FUNCTION_BLOCK orchestratorFB (* Generated orchestrator *)
  (* Standard: 61499-2 *)
  (* Version 1.0, 2020-10-07, generator *)
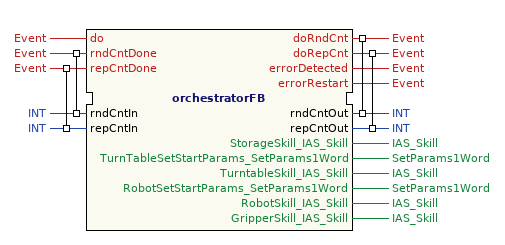
  EVENT_INPUT
    do; (* Start whole process *)
    rndCntDone WITH rndCntIn; (* Whole process (round) counter was updated *)
    repCntDone WITH repCntIn; (* Repetition counter was updated *)
  END_EVENT
  EVENT_OUTPUT
    doRndCnt WITH rndCntOut; (* Update of the whole process (round) counter *)
    doRepCnt WITH repCntOut; (* Update of the repetition counter *)
    errorDetected; (* Triggered when an error signal was received (defined by adapter service sequence) *)
    errorRestart; (* Triggered when error handling and skill restart is started after error signal *)
  END_EVENT
  VAR_INPUT
    rndCntIn : INT; (* Iteration number of the whole process (round) *)
    repCntIn : INT; (* Iteration number of the current repetition process *)
  END_VAR
  VAR_OUTPUT
    rndCntOut : INT; (* Iteration number of the whole process (round) *)
    repCntOut : INT; (* Iteration number of the current repetition process *)
  END_VAR
  PLUGS
    StorageSkill_IAS_Skill : IAS_Skill;
    TurnTableSetStartParams_SetParams1Word : SetParams1Word;
    TurntableSkill_IAS_Skill : IAS_Skill;
    RobotSetStartParams_SetParams1Word : SetParams1Word;
    RobotSkill_IAS_Skill : IAS_Skill;
    GripperSkill_IAS_Skill : IAS_Skill;
  END_PLUGS
  EC_STATES
    START; (* Initial State *)
    Init : round_cnt_reset -> doRndCnt; (* If the adapter of a skill needs an initialization call *)
    Round_Start; (* Start of an iteration of the whole process *)
    Round_End : round_cnt_inc -> doRndCnt; (* End of an iteration of the whole process *)
    0_StorageSkill_Start_0 : -> StorageSkill_IAS_Skill.start;
    1_StorageSkill_RSP_rec_0;
    3_StorageSkill_End_0;
    5_TurnTableSetStartParams_End_1 : 4_TurnTableSetStartParams_Start_1_Alg0 -> TurnTableSetStartParams_SetParams1Word.IND;
    6_TurntableSkill_Start_2 : -> TurntableSkill_IAS_Skill.start;
    7_TurntableSkill_RSP_rec_2;
    9_TurntableSkill_End_2;
    10_StorageSkill_Start_3 : -> StorageSkill_IAS_Skill.start;
    11_StorageSkill_RSP_rec_3;
    13_StorageSkill_End_3;
    15_TurnTableSetStartParams_End_4 : 14_TurnTableSetStartParams_Start_4_Alg1 -> TurnTableSetStartParams_SetParams1Word.IND;
    16_TurntableSkill_Start_5 : -> TurntableSkill_IAS_Skill.start;
    17_TurntableSkill_RSP_rec_5;
    19_TurntableSkill_End_5;
    21_RobotSetStartParams_End_6 : 20_RobotSetStartParams_Start_6_Alg2 -> RobotSetStartParams_SetParams1Word.IND;
    22_RobotSkill_Start_7 : -> RobotSkill_IAS_Skill.start;
    23_RobotSkill_RSP_rec_7;
    25_RobotSkill_End_7;
    26_GripperSkill_Start_8 : -> GripperSkill_IAS_Skill.start;
    27_GripperSkill_RSP_rec_8;
    29_GripperSkill_End_8;
    31_RobotSetStartParams_End_9 : 30_RobotSetStartParams_Start_9_Alg3 -> RobotSetStartParams_SetParams1Word.IND;
    32_RobotSkill_Start_10 : -> RobotSkill_IAS_Skill.start;
    33_RobotSkill_RSP_rec_10;
    35_RobotSkill_End_10;
    36_GripperSkill_Start_11 : -> GripperSkill_IAS_Skill.start;
    37_GripperSkill_RSP_rec_11;
    39_GripperSkill_End_11;
    41_RobotSetStartParams_End_12 : 40_RobotSetStartParams_Start_12_Alg4 -> RobotSetStartParams_SetParams1Word.IND;
    42_RobotSkill_Start_13 : -> RobotSkill_IAS_Skill.start;
    43_RobotSkill_RSP_rec_13;
    45_RobotSkill_End_13;
    46_GripperSkill_Start_14 : -> GripperSkill_IAS_Skill.start;
    47_GripperSkill_RSP_rec_14;
    49_GripperSkill_End_14;
    51_RobotSetStartParams_End_15 : 50_RobotSetStartParams_Start_15_Alg5 -> RobotSetStartParams_SetParams1Word.IND;
    52_RobotSkill_Start_16 : -> RobotSkill_IAS_Skill.start;
    53_RobotSkill_RSP_rec_16;
    55_RobotSkill_End_16;
    56_GripperSkill_Start_17 : -> GripperSkill_IAS_Skill.start;
    57_GripperSkill_RSP_rec_17;
    59_GripperSkill_End_17;
    61_RobotSetStartParams_End_18 : 60_RobotSetStartParams_Start_18_Alg6 -> RobotSetStartParams_SetParams1Word.IND;
    62_RobotSkill_Start_19 : -> RobotSkill_IAS_Skill.start;
    63_RobotSkill_RSP_rec_19;
    65_RobotSkill_End_19;
    66_GripperSkill_Start_20 : -> GripperSkill_IAS_Skill.start;
    67_GripperSkill_RSP_rec_20;
    69_GripperSkill_End_20;
    71_RobotSetStartParams_End_21 : 70_RobotSetStartParams_Start_21_Alg7 -> RobotSetStartParams_SetParams1Word.IND;
    72_RobotSkill_Start_22 : -> RobotSkill_IAS_Skill.start;
    73_RobotSkill_RSP_rec_22;
    75_RobotSkill_End_22;
    76_GripperSkill_Start_23 : -> GripperSkill_IAS_Skill.start;
    77_GripperSkill_RSP_rec_23;
    79_GripperSkill_End_23;
    81_RobotSetStartParams_End_24 : 80_RobotSetStartParams_Start_24_Alg8 -> RobotSetStartParams_SetParams1Word.IND;
    82_RobotSkill_Start_25 : -> RobotSkill_IAS_Skill.start;
    83_RobotSkill_RSP_rec_25;
    85_RobotSkill_End_25;
    86_GripperSkill_Start_26 : -> GripperSkill_IAS_Skill.start;
    87_GripperSkill_RSP_rec_26;
    89_GripperSkill_End_26;
    91_RobotSetStartParams_End_27 : 90_RobotSetStartParams_Start_27_Alg9 -> RobotSetStartParams_SetParams1Word.IND;
    92_RobotSkill_Start_28 : -> RobotSkill_IAS_Skill.start;
    93_RobotSkill_RSP_rec_28;
    95_RobotSkill_End_28;
    96_GripperSkill_Start_29 : -> GripperSkill_IAS_Skill.start;
    97_GripperSkill_RSP_rec_29;
    99_GripperSkill_End_29;
    101_RobotSetStartParams_End_30 : 100_RobotSetStartParams_Start_30_Alg10 -> RobotSetStartParams_SetParams1Word.IND;
    102_RobotSkill_Start_31 : -> RobotSkill_IAS_Skill.start;
    103_RobotSkill_RSP_rec_31;
    105_RobotSkill_End_31;
  END_STATES
  EC_TRANSITIONS
    START TO Init := do;
    Init TO Round_Start := 1;
    Round_End TO Round_Start := do;
    Round_Start TO 0_StorageSkill_Start_0 := 1;
    105_RobotSkill_End_31 TO Round_End := 1;
    0_StorageSkill_Start_0 TO 1_StorageSkill_RSP_rec_0 := StorageSkill_IAS_Skill.RSP[StorageSkill_IAS_Skill.currentState="Executing"];
    1_StorageSkill_RSP_rec_0 TO 3_StorageSkill_End_0 := StorageSkill_IAS_Skill.RSP[StorageSkill_IAS_Skill.currentState="Idle"];
    3_StorageSkill_End_0 TO 5_TurnTableSetStartParams_End_1 := 1;
    5_TurnTableSetStartParams_End_1 TO 6_TurntableSkill_Start_2 := 1;
    6_TurntableSkill_Start_2 TO 7_TurntableSkill_RSP_rec_2 := TurntableSkill_IAS_Skill.RSP[TurntableSkill_IAS_Skill.currentState="Executing"];
    7_TurntableSkill_RSP_rec_2 TO 9_TurntableSkill_End_2 := TurntableSkill_IAS_Skill.RSP[TurntableSkill_IAS_Skill.currentState="Idle"];
    9_TurntableSkill_End_2 TO 10_StorageSkill_Start_3 := 1;
    10_StorageSkill_Start_3 TO 11_StorageSkill_RSP_rec_3 := StorageSkill_IAS_Skill.RSP[StorageSkill_IAS_Skill.currentState="Executing"];
    11_StorageSkill_RSP_rec_3 TO 13_StorageSkill_End_3 := StorageSkill_IAS_Skill.RSP[StorageSkill_IAS_Skill.currentState="Idle"];
    13_StorageSkill_End_3 TO 15_TurnTableSetStartParams_End_4 := 1;
    15_TurnTableSetStartParams_End_4 TO 16_TurntableSkill_Start_5 := 1;
    16_TurntableSkill_Start_5 TO 17_TurntableSkill_RSP_rec_5 := TurntableSkill_IAS_Skill.RSP[TurntableSkill_IAS_Skill.currentState="Executing"];
    17_TurntableSkill_RSP_rec_5 TO 19_TurntableSkill_End_5 := TurntableSkill_IAS_Skill.RSP[TurntableSkill_IAS_Skill.currentState="Idle"];
    19_TurntableSkill_End_5 TO 21_RobotSetStartParams_End_6 := 1;
    21_RobotSetStartParams_End_6 TO 22_RobotSkill_Start_7 := 1;
    22_RobotSkill_Start_7 TO 23_RobotSkill_RSP_rec_7 := RobotSkill_IAS_Skill.RSP[RobotSkill_IAS_Skill.currentState="Executing"];
    23_RobotSkill_RSP_rec_7 TO 25_RobotSkill_End_7 := RobotSkill_IAS_Skill.RSP[RobotSkill_IAS_Skill.currentState="Idle"];
    25_RobotSkill_End_7 TO 26_GripperSkill_Start_8 := 1;
    26_GripperSkill_Start_8 TO 27_GripperSkill_RSP_rec_8 := GripperSkill_IAS_Skill.RSP[GripperSkill_IAS_Skill.currentState="Executing"];
    27_GripperSkill_RSP_rec_8 TO 29_GripperSkill_End_8 := GripperSkill_IAS_Skill.RSP[GripperSkill_IAS_Skill.currentState="Idle"];
    29_GripperSkill_End_8 TO 31_RobotSetStartParams_End_9 := 1;
    31_RobotSetStartParams_End_9 TO 32_RobotSkill_Start_10 := 1;
    32_RobotSkill_Start_10 TO 33_RobotSkill_RSP_rec_10 := RobotSkill_IAS_Skill.RSP[RobotSkill_IAS_Skill.currentState="Executing"];
    33_RobotSkill_RSP_rec_10 TO 35_RobotSkill_End_10 := RobotSkill_IAS_Skill.RSP[RobotSkill_IAS_Skill.currentState="Idle"];
    35_RobotSkill_End_10 TO 36_GripperSkill_Start_11 := 1;
    36_GripperSkill_Start_11 TO 37_GripperSkill_RSP_rec_11 := GripperSkill_IAS_Skill.RSP[GripperSkill_IAS_Skill.currentState="Executing"];
    37_GripperSkill_RSP_rec_11 TO 39_GripperSkill_End_11 := GripperSkill_IAS_Skill.RSP[GripperSkill_IAS_Skill.currentState="Idle"];
    39_GripperSkill_End_11 TO 41_RobotSetStartParams_End_12 := 1;
    41_RobotSetStartParams_End_12 TO 42_RobotSkill_Start_13 := 1;
    42_RobotSkill_Start_13 TO 43_RobotSkill_RSP_rec_13 := RobotSkill_IAS_Skill.RSP[RobotSkill_IAS_Skill.currentState="Executing"];
    43_RobotSkill_RSP_rec_13 TO 45_RobotSkill_End_13 := RobotSkill_IAS_Skill.RSP[RobotSkill_IAS_Skill.currentState="Idle"];
    45_RobotSkill_End_13 TO 46_GripperSkill_Start_14 := 1;
    46_GripperSkill_Start_14 TO 47_GripperSkill_RSP_rec_14 := GripperSkill_IAS_Skill.RSP[GripperSkill_IAS_Skill.currentState="Executing"];
    47_GripperSkill_RSP_rec_14 TO 49_GripperSkill_End_14 := GripperSkill_IAS_Skill.RSP[GripperSkill_IAS_Skill.currentState="Idle"];
    49_GripperSkill_End_14 TO 51_RobotSetStartParams_End_15 := 1;
    51_RobotSetStartParams_End_15 TO 52_RobotSkill_Start_16 := 1;
    52_RobotSkill_Start_16 TO 53_RobotSkill_RSP_rec_16 := RobotSkill_IAS_Skill.RSP[RobotSkill_IAS_Skill.currentState="Executing"];
    53_RobotSkill_RSP_rec_16 TO 55_RobotSkill_End_16 := RobotSkill_IAS_Skill.RSP[RobotSkill_IAS_Skill.currentState="Idle"];
    55_RobotSkill_End_16 TO 56_GripperSkill_Start_17 := 1;
    56_GripperSkill_Start_17 TO 57_GripperSkill_RSP_rec_17 := GripperSkill_IAS_Skill.RSP[GripperSkill_IAS_Skill.currentState="Executing"];
    57_GripperSkill_RSP_rec_17 TO 59_GripperSkill_End_17 := GripperSkill_IAS_Skill.RSP[GripperSkill_IAS_Skill.currentState="Idle"];
    59_GripperSkill_End_17 TO 61_RobotSetStartParams_End_18 := 1;
    61_RobotSetStartParams_End_18 TO 62_RobotSkill_Start_19 := 1;
    62_RobotSkill_Start_19 TO 63_RobotSkill_RSP_rec_19 := RobotSkill_IAS_Skill.RSP[RobotSkill_IAS_Skill.currentState="Executing"];
    63_RobotSkill_RSP_rec_19 TO 65_RobotSkill_End_19 := RobotSkill_IAS_Skill.RSP[RobotSkill_IAS_Skill.currentState="Idle"];
    65_RobotSkill_End_19 TO 66_GripperSkill_Start_20 := 1;
    66_GripperSkill_Start_20 TO 67_GripperSkill_RSP_rec_20 := GripperSkill_IAS_Skill.RSP[GripperSkill_IAS_Skill.currentState="Executing"];
    67_GripperSkill_RSP_rec_20 TO 69_GripperSkill_End_20 := GripperSkill_IAS_Skill.RSP[GripperSkill_IAS_Skill.currentState="Idle"];
    69_GripperSkill_End_20 TO 71_RobotSetStartParams_End_21 := 1;
    71_RobotSetStartParams_End_21 TO 72_RobotSkill_Start_22 := 1;
    72_RobotSkill_Start_22 TO 73_RobotSkill_RSP_rec_22 := RobotSkill_IAS_Skill.RSP[RobotSkill_IAS_Skill.currentState="Executing"];
    73_RobotSkill_RSP_rec_22 TO 75_RobotSkill_End_22 := RobotSkill_IAS_Skill.RSP[RobotSkill_IAS_Skill.currentState="Idle"];
    75_RobotSkill_End_22 TO 76_GripperSkill_Start_23 := 1;
    76_GripperSkill_Start_23 TO 77_GripperSkill_RSP_rec_23 := GripperSkill_IAS_Skill.RSP[GripperSkill_IAS_Skill.currentState="Executing"];
    77_GripperSkill_RSP_rec_23 TO 79_GripperSkill_End_23 := GripperSkill_IAS_Skill.RSP[GripperSkill_IAS_Skill.currentState="Idle"];
    79_GripperSkill_End_23 TO 81_RobotSetStartParams_End_24 := 1;
    81_RobotSetStartParams_End_24 TO 82_RobotSkill_Start_25 := 1;
    82_RobotSkill_Start_25 TO 83_RobotSkill_RSP_rec_25 := RobotSkill_IAS_Skill.RSP[RobotSkill_IAS_Skill.currentState="Executing"];
    83_RobotSkill_RSP_rec_25 TO 85_RobotSkill_End_25 := RobotSkill_IAS_Skill.RSP[RobotSkill_IAS_Skill.currentState="Idle"];
    85_RobotSkill_End_25 TO 86_GripperSkill_Start_26 := 1;
    86_GripperSkill_Start_26 TO 87_GripperSkill_RSP_rec_26 := GripperSkill_IAS_Skill.RSP[GripperSkill_IAS_Skill.currentState="Executing"];
    87_GripperSkill_RSP_rec_26 TO 89_GripperSkill_End_26 := GripperSkill_IAS_Skill.RSP[GripperSkill_IAS_Skill.currentState="Idle"];
    89_GripperSkill_End_26 TO 91_RobotSetStartParams_End_27 := 1;
    91_RobotSetStartParams_End_27 TO 92_RobotSkill_Start_28 := 1;
    92_RobotSkill_Start_28 TO 93_RobotSkill_RSP_rec_28 := RobotSkill_IAS_Skill.RSP[RobotSkill_IAS_Skill.currentState="Executing"];
    93_RobotSkill_RSP_rec_28 TO 95_RobotSkill_End_28 := RobotSkill_IAS_Skill.RSP[RobotSkill_IAS_Skill.currentState="Idle"];
    95_RobotSkill_End_28 TO 96_GripperSkill_Start_29 := 1;
    96_GripperSkill_Start_29 TO 97_GripperSkill_RSP_rec_29 := GripperSkill_IAS_Skill.RSP[GripperSkill_IAS_Skill.currentState="Executing"];
    97_GripperSkill_RSP_rec_29 TO 99_GripperSkill_End_29 := GripperSkill_IAS_Skill.RSP[GripperSkill_IAS_Skill.currentState="Idle"];
    99_GripperSkill_End_29 TO 101_RobotSetStartParams_End_30 := 1;
    101_RobotSetStartParams_End_30 TO 102_RobotSkill_Start_31 := 1;
    102_RobotSkill_Start_31 TO 103_RobotSkill_RSP_rec_31 := RobotSkill_IAS_Skill.RSP[RobotSkill_IAS_Skill.currentState="Executing"];
    103_RobotSkill_RSP_rec_31 TO 105_RobotSkill_End_31 := RobotSkill_IAS_Skill.RSP[RobotSkill_IAS_Skill.currentState="Idle"];
  END_TRANSITIONS
  ALGORITHM round_cnt_inc IN ST: (* Increments the round counter *)
rndCntOut:=rndCntIn+1;
  END_ALGORITHM
  ALGORITHM round_cnt_reset IN ST: (* Resets the round counter *)
rndCntOut:=0;
  END_ALGORITHM
  ALGORITHM rep_cnt_inc IN ST: (* Increments the repetition counter *)
repCntOut:=repCntIn+1;
  END_ALGORITHM
  ALGORITHM rep_cnt_reset IN ST: (* Resets the repetition counter *)
repCntOut:=0;
  END_ALGORITHM
  ALGORITHM 4_TurnTableSetStartParams_Start_1_Alg0 IN ST:
TurnTableSetStartParams_SetParams1Word.DATA:=1;
  END_ALGORITHM
  ALGORITHM 14_TurnTableSetStartParams_Start_4_Alg1 IN ST:
TurnTableSetStartParams_SetParams1Word.DATA:=1;
  END_ALGORITHM
  ALGORITHM 20_RobotSetStartParams_Start_6_Alg2 IN ST:
RobotSetStartParams_SetParams1Word.DATA:=1;
  END_ALGORITHM
  ALGORITHM 30_RobotSetStartParams_Start_9_Alg3 IN ST:
RobotSetStartParams_SetParams1Word.DATA:=1;
  END_ALGORITHM
  ALGORITHM 40_RobotSetStartParams_Start_12_Alg4 IN ST:
RobotSetStartParams_SetParams1Word.DATA:=1;
  END_ALGORITHM
  ALGORITHM 50_RobotSetStartParams_Start_15_Alg5 IN ST:
RobotSetStartParams_SetParams1Word.DATA:=1;
  END_ALGORITHM
  ALGORITHM 60_RobotSetStartParams_Start_18_Alg6 IN ST:
RobotSetStartParams_SetParams1Word.DATA:=1;
  END_ALGORITHM
  ALGORITHM 70_RobotSetStartParams_Start_21_Alg7 IN ST:
RobotSetStartParams_SetParams1Word.DATA:=1;
  END_ALGORITHM
  ALGORITHM 80_RobotSetStartParams_Start_24_Alg8 IN ST:
RobotSetStartParams_SetParams1Word.DATA:=1;
  END_ALGORITHM
  ALGORITHM 90_RobotSetStartParams_Start_27_Alg9 IN ST:
RobotSetStartParams_SetParams1Word.DATA:=1;
  END_ALGORITHM
  ALGORITHM 100_RobotSetStartParams_Start_30_Alg10 IN ST:
RobotSetStartParams_SetParams1Word.DATA:=1;
  END_ALGORITHM
END_FUNCTION_BLOCK
